// TIA Portal project "Elevador" (V17)

(* hardware
DEVICE "S7-1500/ET200MP station_1"  S7-1500 station
   slot 0: "Rail_0"  Rack  6ES7 590-1***0-0AA0
   slot 1: "PLC_1"  CPU 1511-1 PN  6ES7 511-1AK02-0AB0  V2.9
      slot 3: "CPU display_1"  6ES7591-1AA00-0AA0
      slot 32768: "PROFINET interface_1"  X1
         slot 32769: "Port_1"  X1 P1
         slot 32770: "Port_2"  X1 P2
      slot 34817: "Virtual CP interface port_1"  Virtual CP interface port  Virtual CP interface port
*)

// ===== PLC "PLC_1"  CPU 1511-1 PN =====

VAR_GLOBAL   // PLC tag table "Default tag table"
   "BP1" AT %I0.0 : Bool;   // Boton subir elevador
   "BP2" AT %I0.1 : Bool;   // Boton bajar elevador
   "LS1" AT %I0.2 : Bool;   // Limite piso inferior (cocina)
   "LS2" AT %I0.3 : Bool;   // Limite piso superior (servicio)
   "MC1" AT %Q0.0 : Bool;   // Contactor motor subida
   "MC2" AT %Q0.1 : Bool;   // Contactor motor bajada
   "L1" AT %Q0.2 : Bool;   // Lampara piso inferior
   "L2" AT %Q0.3 : Bool;   // Lampara piso superior
END_VAR

TYPE "struct_Elevator_Interface"
   STRUCT
      BP1 : Bool;   // Boton subir
      BP2 : Bool;   // Boton bajar
      LS1 : Bool;   // Limite inferior (cocina)
      LS2 : Bool;   // Limite superior (servicio)
      MC1 : Bool;   // Contactor subida
      MC2 : Bool;   // Contactor bajada
      L1 : Bool;   // Lampara piso inferior
      L2 : Bool;   // Lampara piso superior
   END_STRUCT;
END_TYPE

DATA_BLOCK "DB_Elevador_Interface"   // DB1
{ S7_Optimized_Access := 'FALSE' }
VERSION : 0.1
   VAR
      Interface : "struct_Elevator_Interface";
   END_VAR
BEGIN
END_DATA_BLOCK

DATA_BLOCK "FB_Elevator_Enterprise_DB"   // DB2
{ S7_Optimized_Access := 'TRUE' }
VERSION : 0.1
// stored: InstanceOfName FB_Elevator_Enterprise
"FB_Elevator_Enterprise"
BEGIN
END_DATA_BLOCK

FUNCTION_BLOCK "FB_Elevator_Enterprise"   // FB1, SCL
{ S7_Optimized_Access := 'TRUE' }
VERSION : 0.1
   VAR
      State_Up : Bool;
      State_Down : Bool;
   END_VAR
BEGIN
   // -------------------------
   // INDICADORES DE POSICION
   // -------------------------
   "DB_Elevador_Interface".Interface.L1 := "DB_Elevador_Interface".Interface.LS1;
   "DB_Elevador_Interface".Interface.L2 := "DB_Elevador_Interface".Interface.LS2;

   // -------------------------
   // LOGICA DE SUBIDA
   // -------------------------
   IF "DB_Elevador_Interface".Interface.BP1 AND "DB_Elevador_Interface".Interface.LS1 AND NOT #State_Down THEN
       #State_Up := TRUE;
   END_IF;

   IF "DB_Elevador_Interface".Interface.LS2 THEN
       #State_Up := FALSE;
   END_IF;

   // -------------------------
   // LOGICA DE BAJADA
   // -------------------------
   IF "DB_Elevador_Interface".Interface.BP2 AND "DB_Elevador_Interface".Interface.LS2 AND NOT #State_Up THEN
       #State_Down := TRUE;
   END_IF;

   IF "DB_Elevador_Interface".Interface.LS1 THEN
       #State_Down := FALSE;
   END_IF;

   // -------------------------
   // SALIDAS A MOTOR
   // -------------------------
   "DB_Elevador_Interface".Interface.MC1 := #State_Up AND NOT "DB_Elevador_Interface".Interface.LS2;
   "DB_Elevador_Interface".Interface.MC2 := #State_Down AND NOT "DB_Elevador_Interface".Interface.LS1;
END_FUNCTION_BLOCK

ORGANIZATION_BLOCK "Main"   // OB1, LAD, ProgramCycle
TITLE = "Main Program Sweep (Cycle)"
{ S7_Optimized_Access := 'TRUE' }
VERSION : 0.1
   VAR_INPUT
      Initial_Call : Bool;   // Initial call of this OB
      Remanence : Bool;   // =True, if remanent data are available
   END_VAR
BEGIN

REGION Network 1
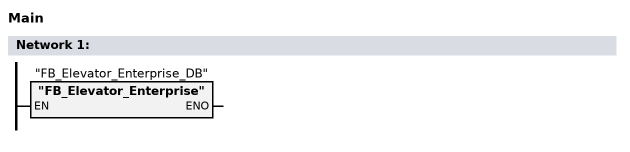
   RUNG wire#powerrail
      "FB_Elevator_Enterprise_DB"()
   END_RUNG
   // the same network as SCL:
   "FB_Elevator_Enterprise_DB"();   // "FB_Elevator_Enterprise"
END_REGION
END_ORGANIZATION_BLOCK